// TIA Portal V17 export
FUNCTION "FC_MainControl" : Void   // FC, LAD
{ S7_Optimized_Access := 'TRUE' }
   VAR_TEMP   // added for the SCL form of the ladder/FBD networks
      _w1 : Bool;
   END_VAR
BEGIN

REGION Network 1: 变频器读取失败上升沿置位
   // 检测"内部数据"."变频器读取失败1"上升沿，置位"内部数据"."变频器通讯故障标志"
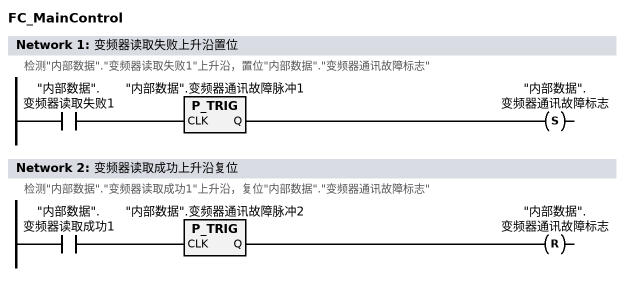
   RUNG wire#powerrail
      Contact( "内部数据".变频器读取失败1 )
      P_Trig( "内部数据".变频器通讯故障脉冲1 )
      S_Coil( "内部数据".变频器通讯故障标志 )
   END_RUNG
   // the same network as SCL:
   #_w1 := "内部数据".变频器读取失败1 AND NOT "内部数据".变频器通讯故障脉冲1;   // rising edge
   "内部数据".变频器通讯故障脉冲1 := "内部数据".变频器读取失败1;
   IF #_w1 THEN "内部数据".变频器通讯故障标志 := TRUE; END_IF;
END_REGION

REGION Network 2: 变频器读取成功上升沿复位
   // 检测"内部数据"."变频器读取成功1"上升沿，复位"内部数据"."变频器通讯故障标志"
   RUNG wire#powerrail
      Contact( "内部数据".变频器读取成功1 )
      P_Trig( "内部数据".变频器通讯故障脉冲2 )
      R_Coil( "内部数据".变频器通讯故障标志 )
   END_RUNG
   // the same network as SCL:
   #_w1 := "内部数据".变频器读取成功1 AND NOT "内部数据".变频器通讯故障脉冲2;   // rising edge
   "内部数据".变频器通讯故障脉冲2 := "内部数据".变频器读取成功1;
   IF #_w1 THEN "内部数据".变频器通讯故障标志 := FALSE; END_IF;
END_REGION
END_FUNCTION
